FUNCTION_BLOCK FB_CartCtrlReady EXTENDS FB_CartCtrlBase
VAR_INPUT
END_VAR
VAR_OUTPUT
END_VAR
VAR
END_VAR

// override this function in each exact controller
METHOD PROTECTED calcCmdJntPos : BOOL
VAR_IN_OUT CONSTANT
	// slave cart joint data
	i_slaveCart :FB_SlaveCart;
END_VAR
//m_cmdJntPos := i_slaveCart.curJntPos;
END_METHOD

// override this function in each exact controller
// NOTICE: set joint control mode here, and do some initialization if needed
METHOD PUBLIC init : BOOL
VAR_IN_OUT CONSTANT
	i_slaveCart	:FB_SlaveCart;
END_VAR
VAR_IN_OUT 
	r_cartCtrlCmd :ST_SlaveArmCtrlCmds;
END_VAR
//m_holdLastCmds := checkToHoldLastCmds(i_slaveCart);
m_holdLastCmds := checkToHoldLastCmds(i_slaveCart);
SUPER^.init(i_slaveCart,r_cartCtrlCmd);
m_cmdJntPos[5]:=i_slaveCart.m_curJntPos[5];
// update commands to arm
copyCmds(r_cartCtrlCmd);
END_METHOD

END_FUNCTION_BLOCK

(* stored: Version 1.1.0.1, ProductVersion 3.1.4024.11
   POU FB_CartCtrlReady: Id {d9e6de9d-36e0-4638-ae50-750334c7fa40}, SpecialFunc None
   Method calcCmdJntPos: Id {76f24731-8ab2-4654-b6a2-22c40abd6854}
   Method init: Id {dfe1fe06-fc95-4692-9cd0-0f60ba7eeb72} *)
